(* Logix 5000 project; controller simulacion1 Emulate 5570 rev 32.11; software revision 32.00 *)

TASK MainTask (continuous, watchdog 500 ms) : MainProgram

MODULES
   Local : Emulate 5570 (ICP 2, rev 32.11)
      I_O : vendor 1 type 0 code 15 (ICP 3, rev 1.1, Output RPI 50 ms)   // modulo de entradas y salidas
END_MODULES

VAR_GLOBAL   (* controller tags *)
   A1 : BOOL;
   M1 : ALIAS FOR Local:3:O.Data[0].0;
   M2 : ALIAS FOR Local:3:O.Data[0].1;
   M3 : ALIAS FOR Local:3:O.Data[0].2;
   S1 : ALIAS FOR Local:3:I.Data[1].0;
   S2 : ALIAS FOR Local:3:I.Data[1].1;
   T1 : TIMER := (PRE := 1000);
END_VAR

PROGRAM MainProgram   (* main routine MainRoutine *)

ROUTINE MainRoutine   (* ladder *)
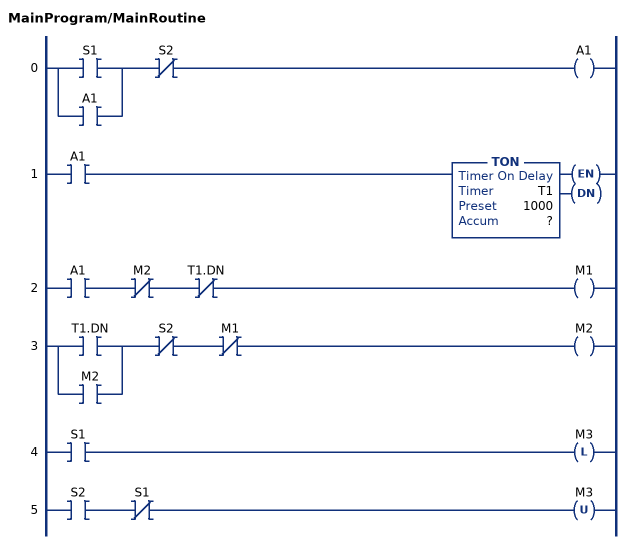
   0: [XIC(S1) ,XIC(A1) ]XIO(S2)OTE(A1);
   1: XIC(A1)TON(T1,?,?);
   2: XIC(A1)XIO(M2)XIO(T1.DN)OTE(M1);
   3: [XIC(T1.DN) ,XIC(M2) ]XIO(S2)XIO(M1)OTE(M2);
   4: XIC(S1)OTL(M3);
   5: XIC(S2)XIO(S1)OTU(M3);
END_ROUTINE
END_PROGRAM
